Universal Robots PolyScope program: VO.urp

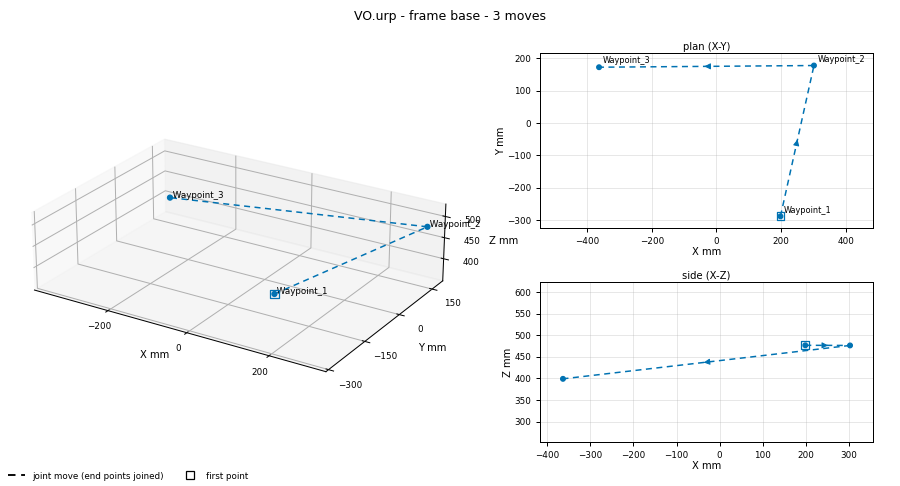
[picture p0: tool path of VO.urp in frame base, 3 of 3 moves have a stored position in this frame; points joined in program order, loops and branches not executed]
Program VO (installation=default directory=/programs/usbdisk/sources createdIn=5.19.0 lastSavedIn=5.19.0 robotSerialNumber=20235366666)
Calibrated DH parameters: a=[-0.000074, -0.240481, -0.025105, 0.000089, -0.000025, 0]; d=[0.151722, 81.163768, -218.075848, 137.042846, 0.08536, 0.091978]; alpha=[1.570306, -0.000479, -0.001547, 1.572519, -1.572356, 0]; deltaTheta=[0, -0.16012, 1.612913, -1.452801, 0, 0]
InitVariablesNode
Robot Program (runOnlyOnce=false)
  MoveL speed 250 mm/s, acceleration 1200 mm/s^2 (useActiveTCP=true) feature=Base
    Waypoint Waypoint_1: TCP in base x=198.442 y=-288.67 z=476.878 mm, rx=0.0462 ry=0.0946 rz=1.9597 rad; joints [101.305, -4.177, -86.816, -0.578, 85.022, 101.208] deg
  MoveJ speed 60 deg/s, acceleration 80 deg/s^2 (useActiveTCP=true) feature=Base
    Waypoint Waypoint_2: TCP in base x=302.116 y=178.23 z=476.578 mm, rx=0.0349 ry=-0.1218 rz=-2.8174 rad; joints [-172.63, -4.136, -86.764, -0.579, 85.019, 101.203] deg
  MoveJ speed 60 deg/s, acceleration 80 deg/s^2 (useActiveTCP=true) feature=Base
    Waypoint Waypoint_3: TCP in base x=-363.135 y=172.999 z=399.196 mm, rx=-0.0063 ry=-2.0709 rz=-2.0847 rad; joints [-171.91, -174.863, 82.693, 189.406, -0.882, -88.889] deg
